FUNCTION_BLOCK FEATURE_EXTRACTION
  {SET_ATTRIBUTE(OpcUa, SERVICE)}
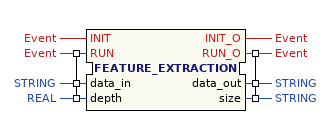
  EVENT_INPUT
    INIT;
    RUN WITH data_in, depth; {SET_ATTRIBUTE(OpcUa, Method)}
  END_EVENT
  EVENT_OUTPUT
    INIT_O;
    RUN_O WITH data_out, size;
  END_EVENT
  VAR_INPUT
    data_in : STRING; {SET_ATTRIBUTE(OpcUa, Variable)}
    depth : REAL; {SET_ATTRIBUTE(OpcUa, Constant)}
  END_VAR
  VAR_OUTPUT
    data_out : STRING; {SET_ATTRIBUTE(OpcUa, Variable)}
    size : STRING; {SET_ATTRIBUTE(OpcUa, Variable)}
  END_VAR
END_FUNCTION_BLOCK
